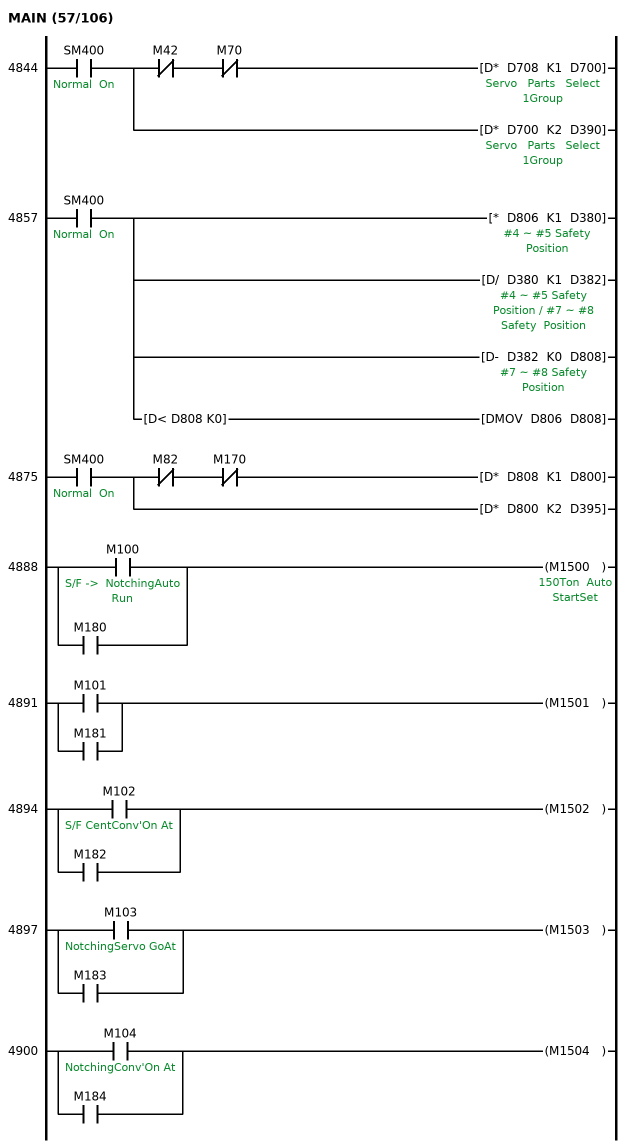
[picture p336: ladder of MAIN, rungs at steps 4844 to 4900]
4844  LD      SM400  ; Normal  On
      MPS
      ANI     M42
      ANI     M70
      D*      D708 K1 D700  ; Servo   Parts   Select  1Group
      MPP
      D*      D700 K2 D390
4857  LD      SM400  ; Normal  On
      *       D806 K1 D380  ; #4 ~ #5 Safety  Position
      D/      D380 K1 D382  ; #7 ~ #8 Safety  Position
      D-      D382 K0 D808
      ANDD<   D808 K0
      DMOV    D806 D808
4875  LD      SM400  ; Normal  On
      MPS
      ANI     M82
      ANI     M170
      D*      D808 K1 D800
      MPP
      D*      D800 K2 D395
4888  LD      M100  ; S/F ->  NotchingAuto Run
      OR      M180
      OUT     M1500  ; 150Ton  Auto    StartSet
4891  LD      M101
      OR      M181
      OUT     M1501
4894  LD      M102  ; S/F CentConv'On At
      OR      M182
      OUT     M1502
4897  LD      M103  ; NotchingServo GoAt
      OR      M183
      OUT     M1503
4900  LD      M104  ; NotchingConv'On At
      OR      M184
      OUT     M1504
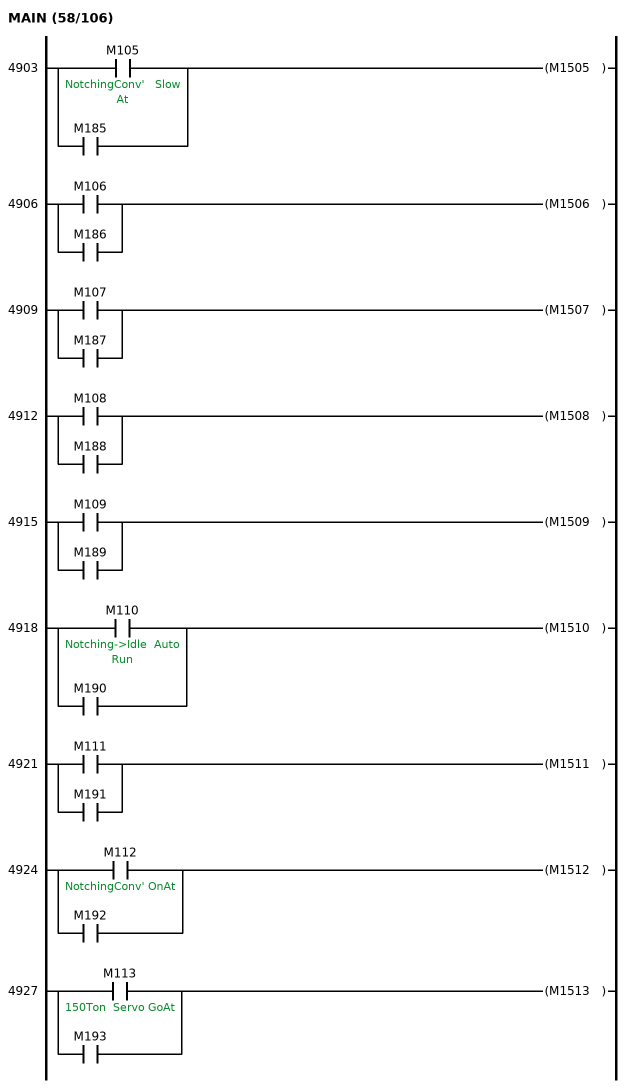
4903  LD      M105  ; NotchingConv'   Slow At
      OR      M185
      OUT     M1505
4906  LD      M106
      OR      M186
      OUT     M1506
4909  LD      M107
      OR      M187
      OUT     M1507
4912  LD      M108
      OR      M188
      OUT     M1508
4915  LD      M109
      OR      M189
      OUT     M1509
4918  LD      M110  ; Notching->Idle  Auto Run
      OR      M190
      OUT     M1510
4921  LD      M111
      OR      M191
      OUT     M1511
4924  LD      M112  ; NotchingConv' OnAt
      OR      M192
      OUT     M1512
4927  LD      M113  ; 150Ton  Servo GoAt
      OR      M193
      OUT     M1513
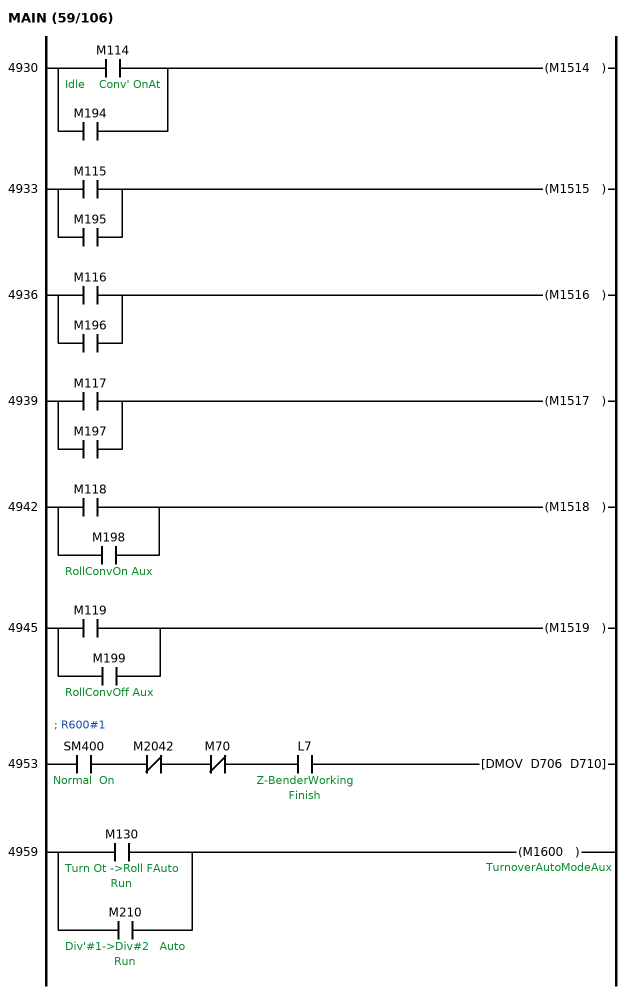
4930  LD      M114  ; Idle    Conv' OnAt
      OR      M194
      OUT     M1514
4933  LD      M115
      OR      M195
      OUT     M1515
4936  LD      M116
      OR      M196
      OUT     M1516
4939  LD      M117
      OR      M197
      OUT     M1517
4942  LD      M118
      OR      M198  ; RollConvOn Aux
      OUT     M1518
4945  LD      M119
      OR      M199  ; RollConvOff Aux
      OUT     M1519
; R600#1
4953  LD      SM400  ; Normal  On
      ANI     M2042
      ANI     M70
      AND     L7  ; Z-BenderWorking Finish
      DMOV    D706 D710
4959  LD      M130  ; Turn Ot ->Roll FAuto Run
      OR      M210  ; Div'#1->Div#2   Auto Run
      OUT     M1600  ; TurnoverAutoModeAux
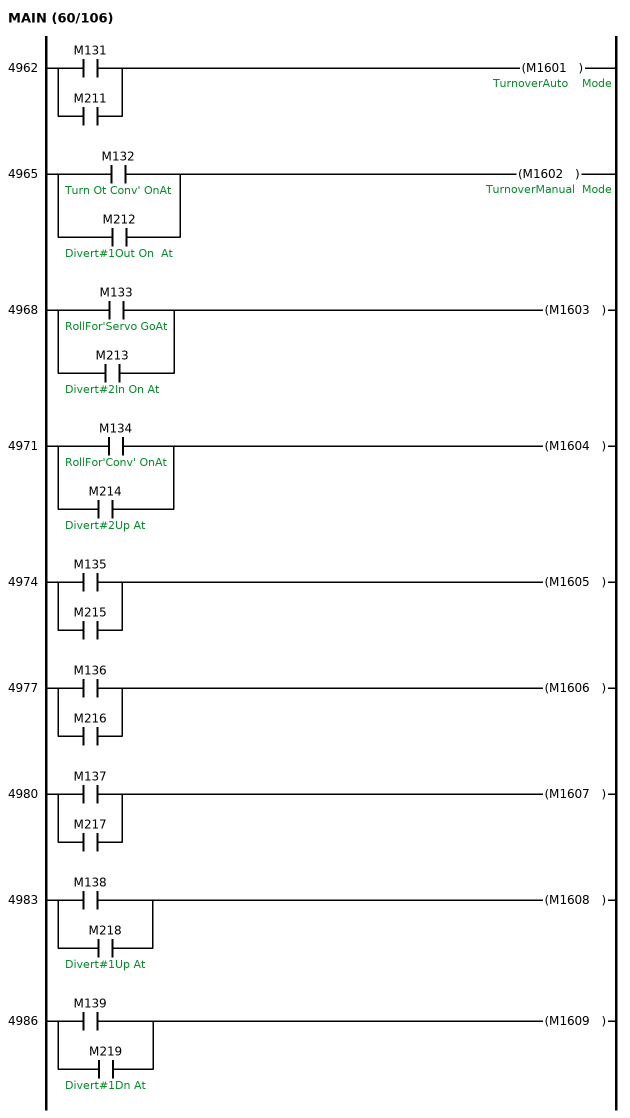
4962  LD      M131
      OR      M211
      OUT     M1601  ; TurnoverAuto    Mode
4965  LD      M132  ; Turn Ot Conv' OnAt
      OR      M212  ; Divert#1Out On  At
      OUT     M1602  ; TurnoverManual  Mode
4968  LD      M133  ; RollFor'Servo GoAt
      OR      M213  ; Divert#2In On At
      OUT     M1603
4971  LD      M134  ; RollFor'Conv' OnAt
      OR      M214  ; Divert#2Up At
      OUT     M1604
4974  LD      M135
      OR      M215
      OUT     M1605
4977  LD      M136
      OR      M216
      OUT     M1606
4980  LD      M137
      OR      M217
      OUT     M1607
4983  LD      M138
      OR      M218  ; Divert#1Up At
      OUT     M1608
4986  LD      M139
      OR      M219  ; Divert#1Dn At
      OUT     M1609
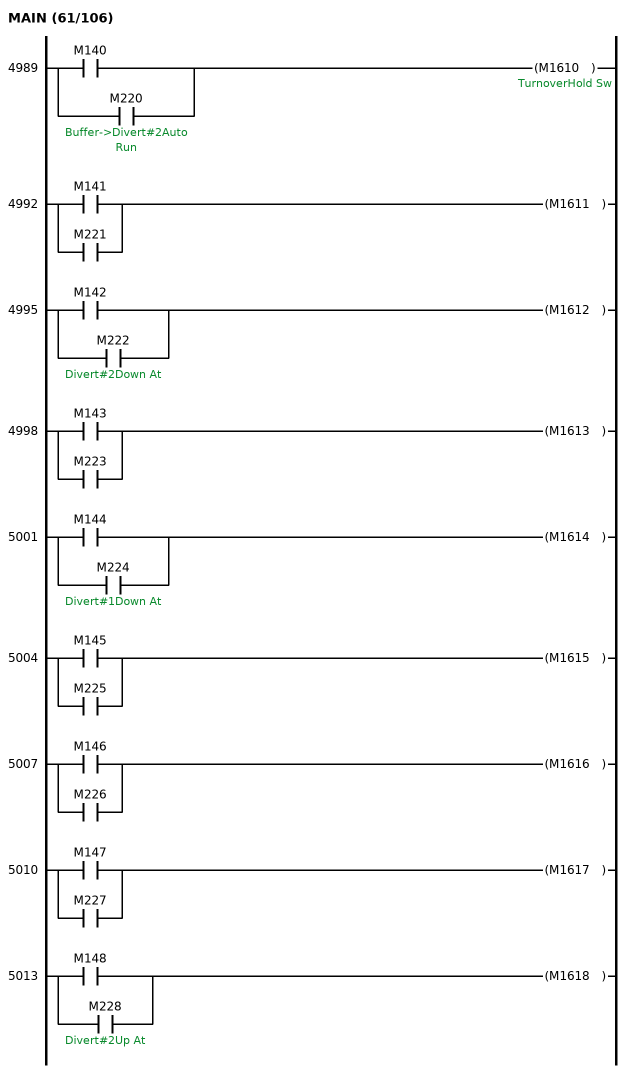
4989  LD      M140
      OR      M220  ; Buffer->Divert#2Auto Run
      OUT     M1610  ; TurnoverHold Sw
4992  LD      M141
      OR      M221
      OUT     M1611
4995  LD      M142
      OR      M222  ; Divert#2Down At
      OUT     M1612
4998  LD      M143
      OR      M223
      OUT     M1613
5001  LD      M144
      OR      M224  ; Divert#1Down At
      OUT     M1614
5004  LD      M145
      OR      M225
      OUT     M1615
5007  LD      M146
      OR      M226
      OUT     M1616
5010  LD      M147
      OR      M227
      OUT     M1617
5013  LD      M148
      OR      M228  ; Divert#2Up At
      OUT     M1618
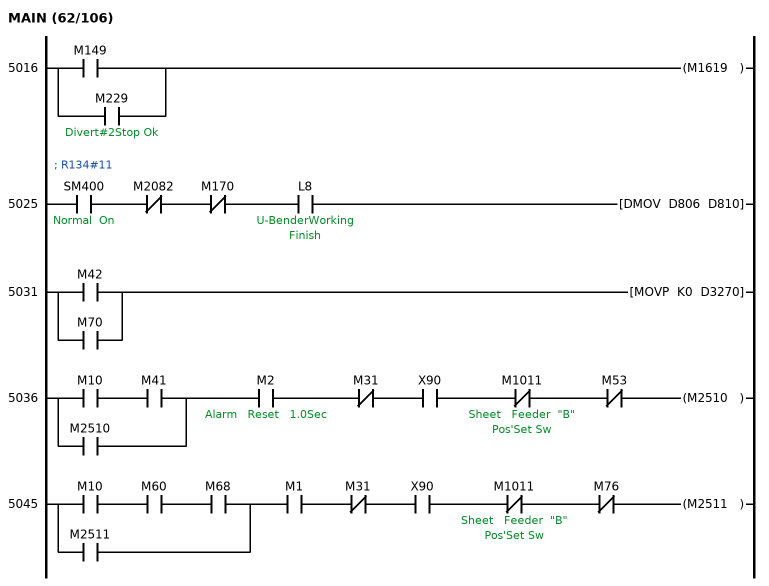
5016  LD      M149
      OR      M229  ; Divert#2Stop Ok
      OUT     M1619
; R134#11
5025  LD      SM400  ; Normal  On
      ANI     M2082
      ANI     M170
      AND     L8  ; U-BenderWorking Finish
      DMOV    D806 D810
5031  LD      M42
      OR      M70
      MOVP    K0 D3270
5036  LD      M10
      AND     M41
      OR      M2510
      AND     M2  ; Alarm   Reset   1.0Sec
      ANI     M31
      AND     X90
      ANI     M1011  ; Sheet   Feeder  "B" Pos'Set Sw
      ANI     M53
      OUT     M2510
5045  LD      M10
      AND     M60
      AND     M68
      OR      M2511
      AND     M1
      ANI     M31
      AND     X90
      ANI     M1011  ; Sheet   Feeder  "B" Pos'Set Sw
      ANI     M76
      OUT     M2511
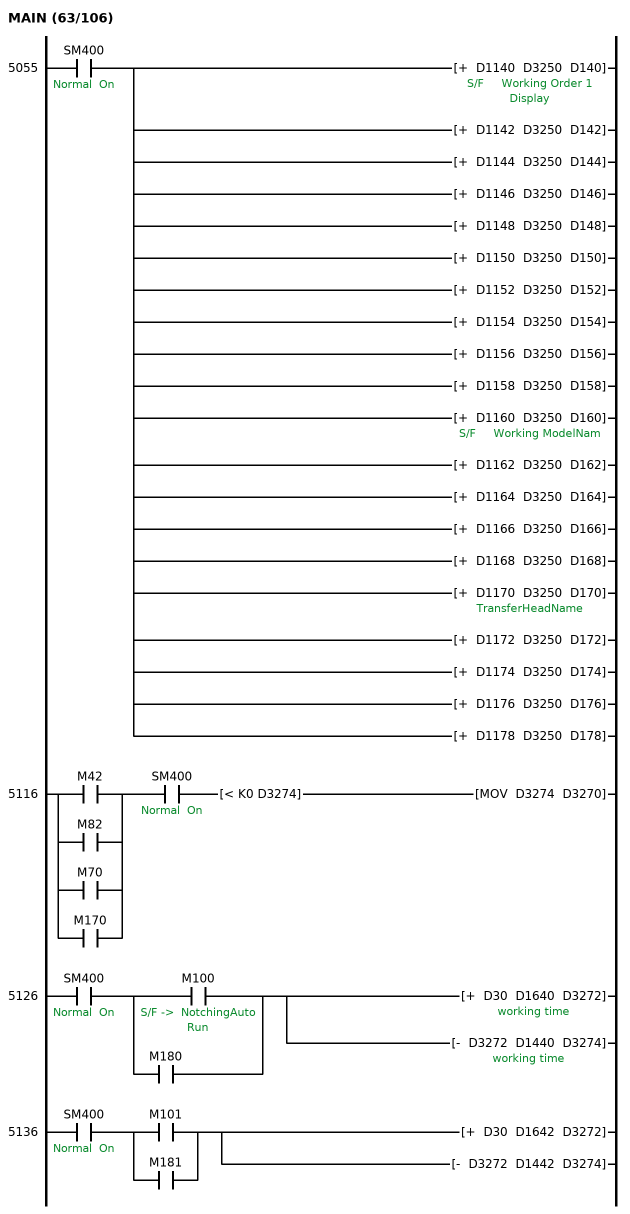
5055  LD      SM400  ; Normal  On
      +       D1140 D3250 D140
      +       D1142 D3250 D142
      +       D1144 D3250 D144
      +       D1146 D3250 D146
      +       D1148 D3250 D148
      +       D1150 D3250 D150
      +       D1152 D3250 D152
      +       D1154 D3250 D154
      +       D1156 D3250 D156
      +       D1158 D3250 D158
      +       D1160 D3250 D160
      +       D1162 D3250 D162
      +       D1164 D3250 D164
      +       D1166 D3250 D166
      +       D1168 D3250 D168
      +       D1170 D3250 D170
      +       D1172 D3250 D172
      +       D1174 D3250 D174
      +       D1176 D3250 D176
      +       D1178 D3250 D178
5116  LD      M42
      OR      M82
      OR      M70
      OR      M170
      AND     SM400  ; Normal  On
      AND<    K0 D3274
      MOV     D3274 D3270
5126  LD      SM400  ; Normal  On
      LD      M100  ; S/F ->  NotchingAuto Run
      OR      M180
      ANB
      +       D30 D1640 D3272  ; working time
      -       D3272 D1440 D3274
5136  LD      SM400  ; Normal  On
      LD      M101
      OR      M181
      ANB
      +       D30 D1642 D3272
      -       D3272 D1442 D3274
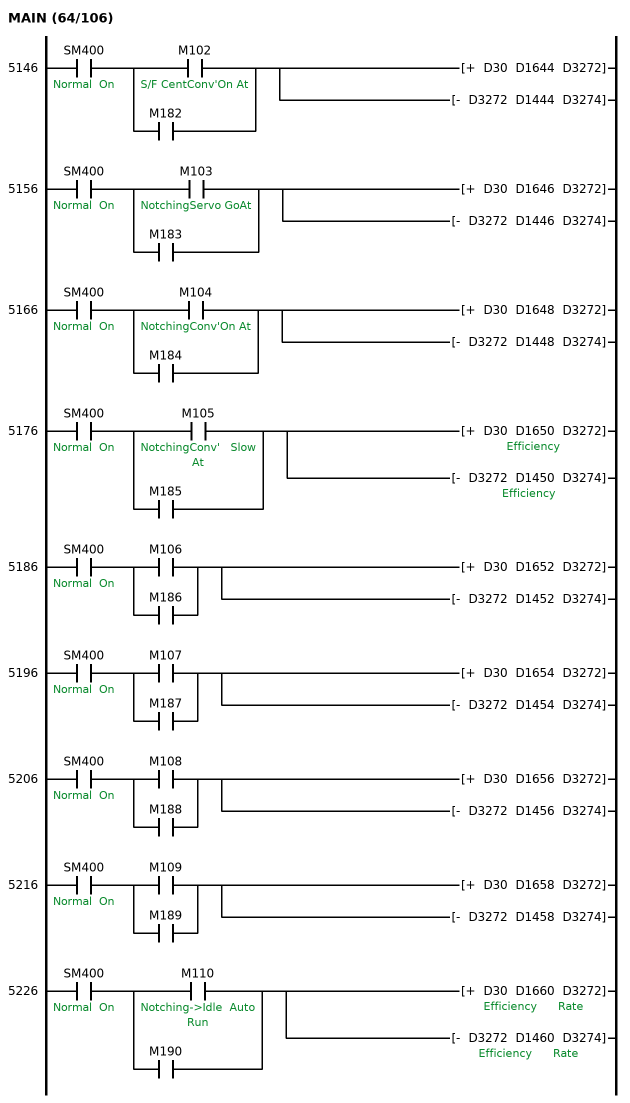
5146  LD      SM400  ; Normal  On
      LD      M102  ; S/F CentConv'On At
      OR      M182
      ANB
      +       D30 D1644 D3272
      -       D3272 D1444 D3274
5156  LD      SM400  ; Normal  On
      LD      M103  ; NotchingServo GoAt
      OR      M183
      ANB
      +       D30 D1646 D3272
      -       D3272 D1446 D3274
5166  LD      SM400  ; Normal  On
      LD      M104  ; NotchingConv'On At
      OR      M184
      ANB
      +       D30 D1648 D3272
      -       D3272 D1448 D3274
5176  LD      SM400  ; Normal  On
      LD      M105  ; NotchingConv'   Slow At
      OR      M185
      ANB
      +       D30 D1650 D3272  ; Efficiency
      -       D3272 D1450 D3274
5186  LD      SM400  ; Normal  On
      LD      M106
      OR      M186
      ANB
      +       D30 D1652 D3272
      -       D3272 D1452 D3274
5196  LD      SM400  ; Normal  On
      LD      M107
      OR      M187
      ANB
      +       D30 D1654 D3272
      -       D3272 D1454 D3274
5206  LD      SM400  ; Normal  On
      LD      M108
      OR      M188
      ANB
      +       D30 D1656 D3272
      -       D3272 D1456 D3274
5216  LD      SM400  ; Normal  On
      LD      M109
      OR      M189
      ANB
      +       D30 D1658 D3272
      -       D3272 D1458 D3274
5226  LD      SM400  ; Normal  On
      LD      M110  ; Notching->Idle  Auto Run
      OR      M190
      ANB
      +       D30 D1660 D3272  ; Efficiency      Rate
      -       D3272 D1460 D3274
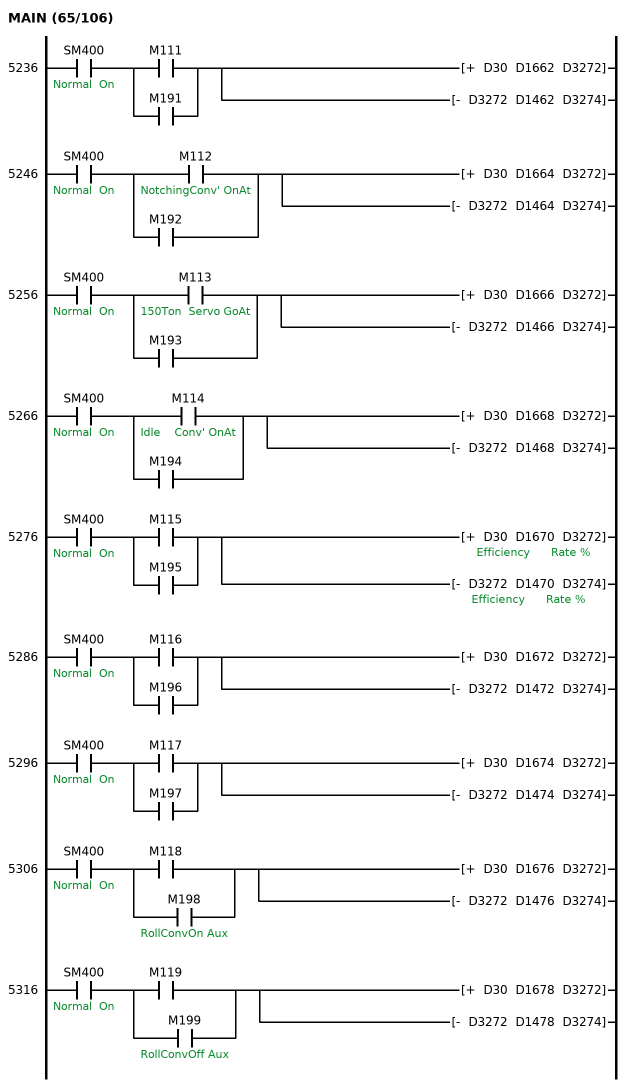
5236  LD      SM400  ; Normal  On
      LD      M111
      OR      M191
      ANB
      +       D30 D1662 D3272
      -       D3272 D1462 D3274
5246  LD      SM400  ; Normal  On
      LD      M112  ; NotchingConv' OnAt
      OR      M192
      ANB
      +       D30 D1664 D3272
      -       D3272 D1464 D3274
5256  LD      SM400  ; Normal  On
      LD      M113  ; 150Ton  Servo GoAt
      OR      M193
      ANB
      +       D30 D1666 D3272
      -       D3272 D1466 D3274
5266  LD      SM400  ; Normal  On
      LD      M114  ; Idle    Conv' OnAt
      OR      M194
      ANB
      +       D30 D1668 D3272
      -       D3272 D1468 D3274
5276  LD      SM400  ; Normal  On
      LD      M115
      OR      M195
      ANB
      +       D30 D1670 D3272  ; Efficiency      Rate %
      -       D3272 D1470 D3274
5286  LD      SM400  ; Normal  On
      LD      M116
      OR      M196
      ANB
      +       D30 D1672 D3272
      -       D3272 D1472 D3274
5296  LD      SM400  ; Normal  On
      LD      M117
      OR      M197
      ANB
      +       D30 D1674 D3272
      -       D3272 D1474 D3274
5306  LD      SM400  ; Normal  On
      LD      M118
      OR      M198  ; RollConvOn Aux
      ANB
      +       D30 D1676 D3272
      -       D3272 D1476 D3274
5316  LD      SM400  ; Normal  On
      LD      M119
      OR      M199  ; RollConvOff Aux
      ANB
      +       D30 D1678 D3272
      -       D3272 D1478 D3274
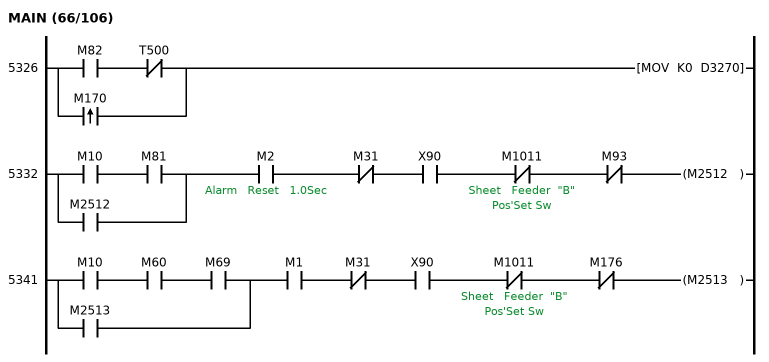
5326  LD      M82
      ANI     T500
      ORP     M170
      MOV     K0 D3270
5332  LD      M10
      AND     M81
      OR      M2512
      AND     M2  ; Alarm   Reset   1.0Sec
      ANI     M31
      AND     X90
      ANI     M1011  ; Sheet   Feeder  "B" Pos'Set Sw
      ANI     M93
      OUT     M2512
5341  LD      M10
      AND     M60
      AND     M69
      OR      M2513
      AND     M1
      ANI     M31
      AND     X90
      ANI     M1011  ; Sheet   Feeder  "B" Pos'Set Sw
      ANI     M176
      OUT     M2513
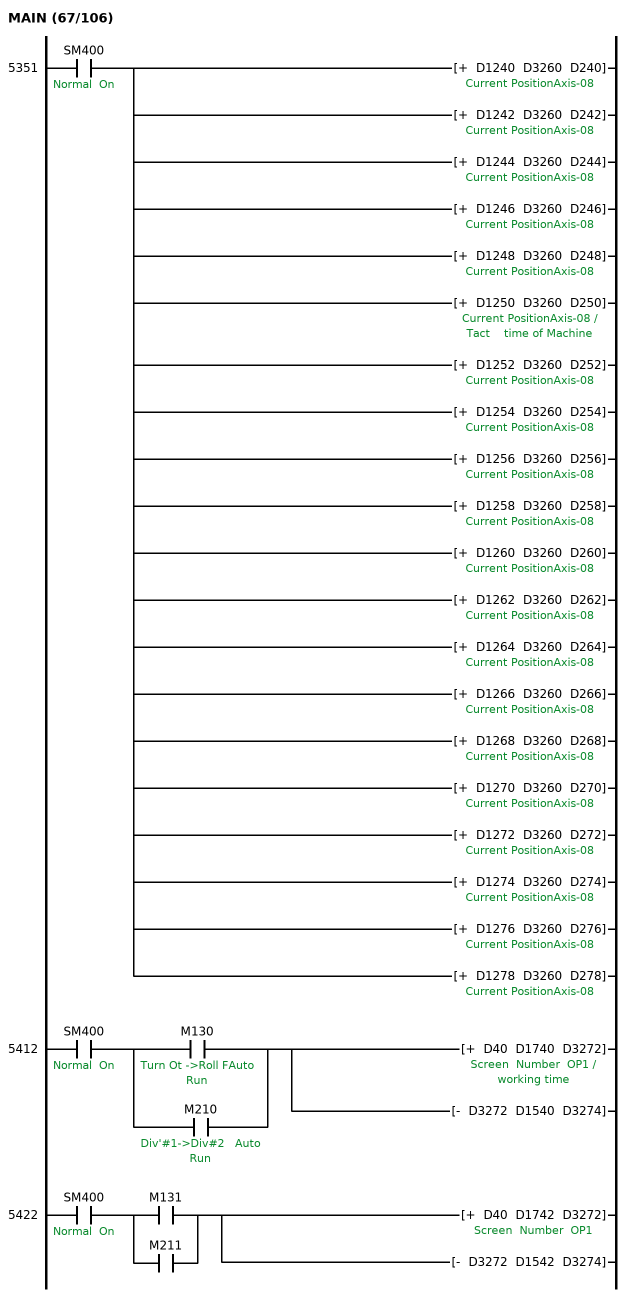
5351  LD      SM400  ; Normal  On
      +       D1240 D3260 D240  ; Current PositionAxis-08
      +       D1242 D3260 D242
      +       D1244 D3260 D244
      +       D1246 D3260 D246
      +       D1248 D3260 D248
      +       D1250 D3260 D250
      +       D1252 D3260 D252
      +       D1254 D3260 D254
      +       D1256 D3260 D256
      +       D1258 D3260 D258
      +       D1260 D3260 D260
      +       D1262 D3260 D262
      +       D1264 D3260 D264
      +       D1266 D3260 D266
      +       D1268 D3260 D268
      +       D1270 D3260 D270
      +       D1272 D3260 D272
      +       D1274 D3260 D274
      +       D1276 D3260 D276
      +       D1278 D3260 D278
5412  LD      SM400  ; Normal  On
      LD      M130  ; Turn Ot ->Roll FAuto Run
      OR      M210  ; Div'#1->Div#2   Auto Run
      ANB
      +       D40 D1740 D3272  ; working time
      -       D3272 D1540 D3274
5422  LD      SM400  ; Normal  On
      LD      M131
      OR      M211
      ANB
      +       D40 D1742 D3272
      -       D3272 D1542 D3274
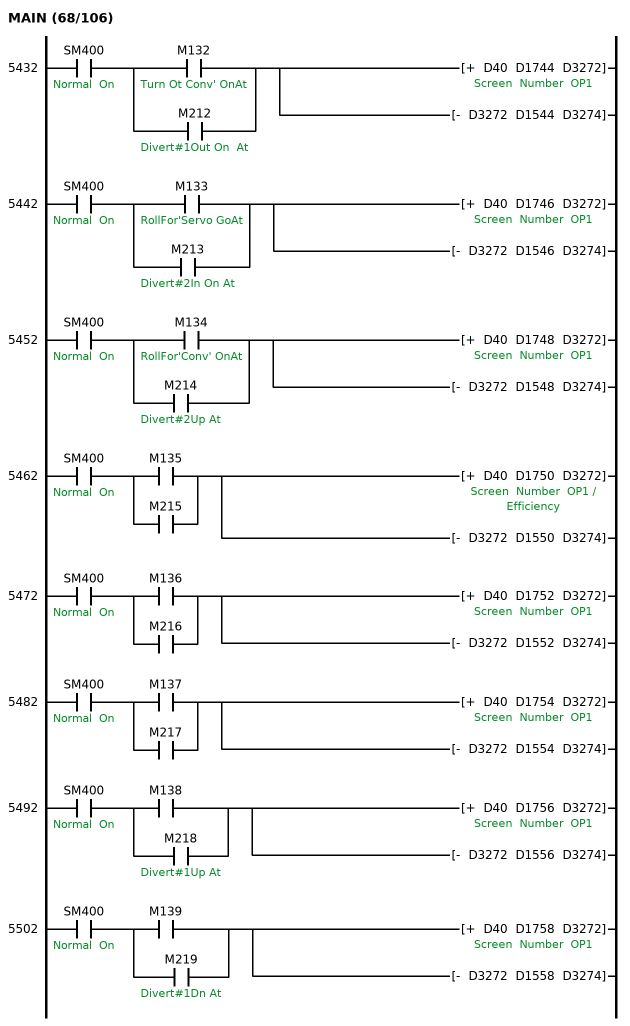
5432  LD      SM400  ; Normal  On
      LD      M132  ; Turn Ot Conv' OnAt
      OR      M212  ; Divert#1Out On  At
      ANB
      +       D40 D1744 D3272
      -       D3272 D1544 D3274
5442  LD      SM400  ; Normal  On
      LD      M133  ; RollFor'Servo GoAt
      OR      M213  ; Divert#2In On At
      ANB
      +       D40 D1746 D3272
      -       D3272 D1546 D3274
5452  LD      SM400  ; Normal  On
      LD      M134  ; RollFor'Conv' OnAt
      OR      M214  ; Divert#2Up At
      ANB
      +       D40 D1748 D3272
      -       D3272 D1548 D3274
5462  LD      SM400  ; Normal  On
      LD      M135
      OR      M215
      ANB
      +       D40 D1750 D3272  ; Efficiency
      -       D3272 D1550 D3274
5472  LD      SM400  ; Normal  On
      LD      M136
      OR      M216
      ANB
      +       D40 D1752 D3272
      -       D3272 D1552 D3274
5482  LD      SM400  ; Normal  On
      LD      M137
      OR      M217
      ANB
      +       D40 D1754 D3272
      -       D3272 D1554 D3274
5492  LD      SM400  ; Normal  On
      LD      M138
      OR      M218  ; Divert#1Up At
      ANB
      +       D40 D1756 D3272
      -       D3272 D1556 D3274
5502  LD      SM400  ; Normal  On
      LD      M139
      OR      M219  ; Divert#1Dn At
      ANB
      +       D40 D1758 D3272
      -       D3272 D1558 D3274
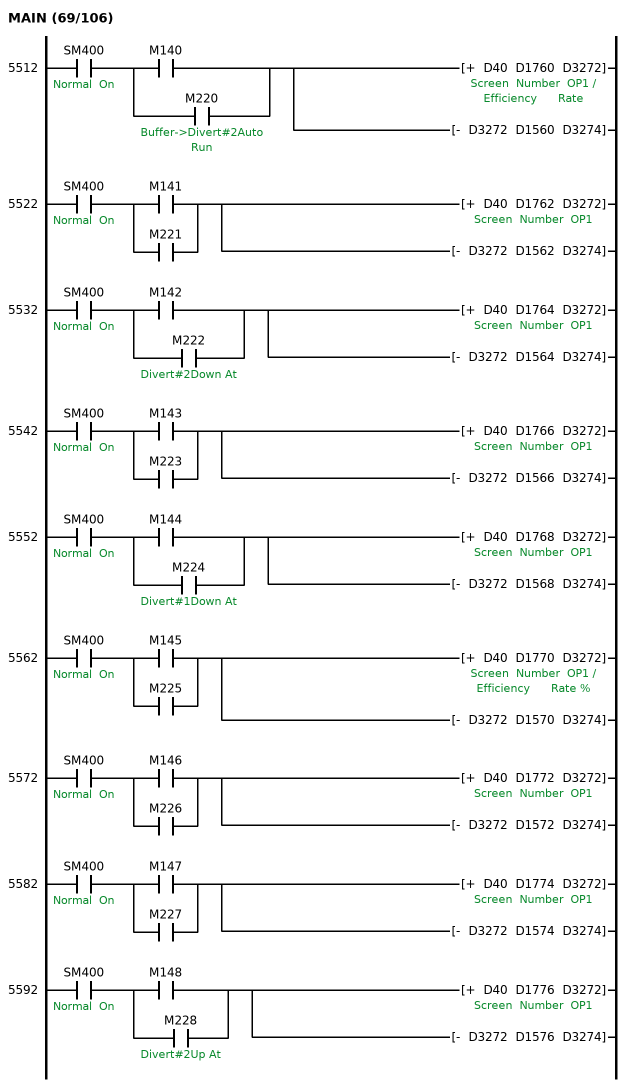
5512  LD      SM400  ; Normal  On
      LD      M140
      OR      M220  ; Buffer->Divert#2Auto Run
      ANB
      +       D40 D1760 D3272  ; Efficiency      Rate
      -       D3272 D1560 D3274
5522  LD      SM400  ; Normal  On
      LD      M141
      OR      M221
      ANB
      +       D40 D1762 D3272
      -       D3272 D1562 D3274
5532  LD      SM400  ; Normal  On
      LD      M142
      OR      M222  ; Divert#2Down At
      ANB
      +       D40 D1764 D3272
      -       D3272 D1564 D3274
5542  LD      SM400  ; Normal  On
      LD      M143
      OR      M223
      ANB
      +       D40 D1766 D3272
      -       D3272 D1566 D3274
5552  LD      SM400  ; Normal  On
      LD      M144
      OR      M224  ; Divert#1Down At
      ANB
      +       D40 D1768 D3272
      -       D3272 D1568 D3274
5562  LD      SM400  ; Normal  On
      LD      M145
      OR      M225
      ANB
      +       D40 D1770 D3272  ; Efficiency      Rate %
      -       D3272 D1570 D3274
5572  LD      SM400  ; Normal  On
      LD      M146
      OR      M226
      ANB
      +       D40 D1772 D3272
      -       D3272 D1572 D3274
5582  LD      SM400  ; Normal  On
      LD      M147
      OR      M227
      ANB
      +       D40 D1774 D3272
      -       D3272 D1574 D3274
5592  LD      SM400  ; Normal  On
      LD      M148
      OR      M228  ; Divert#2Up At
      ANB
      +       D40 D1776 D3272
      -       D3272 D1576 D3274
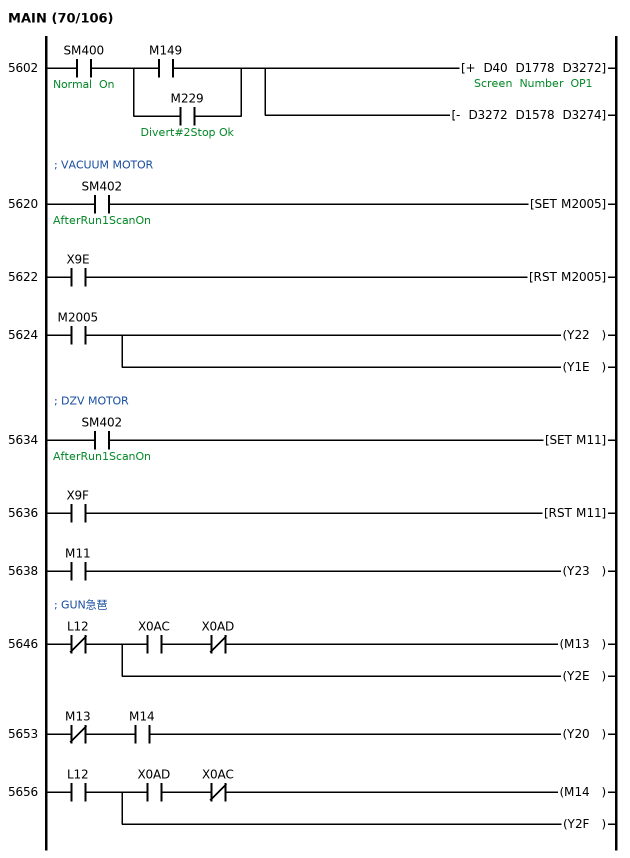
5602  LD      SM400  ; Normal  On
      LD      M149
      OR      M229  ; Divert#2Stop Ok
      ANB
      +       D40 D1778 D3272
      -       D3272 D1578 D3274
; VACUUM MOTOR
5620  LD      SM402  ; AfterRun1ScanOn
      SET     M2005
5622  LD      X9E
      RST     M2005
5624  LD      M2005
      OUT     Y22
      OUT     Y1E
; DZV MOTOR
5634  LD      SM402  ; AfterRun1ScanOn
      SET     M11
5636  LD      X9F
      RST     M11
5638  LD      M11
      OUT     Y23
; GUN선택
5646  LDI     L12
      MPS
      AND     X0AC
      ANI     X0AD
      OUT     M13
      MPP
      OUT     Y2E
5653  LDI     M13
      AND     M14
      OUT     Y20
5656  LD      L12
      MPS
      AND     X0AD
      ANI     X0AC
      OUT     M14
      MPP
      OUT     Y2F
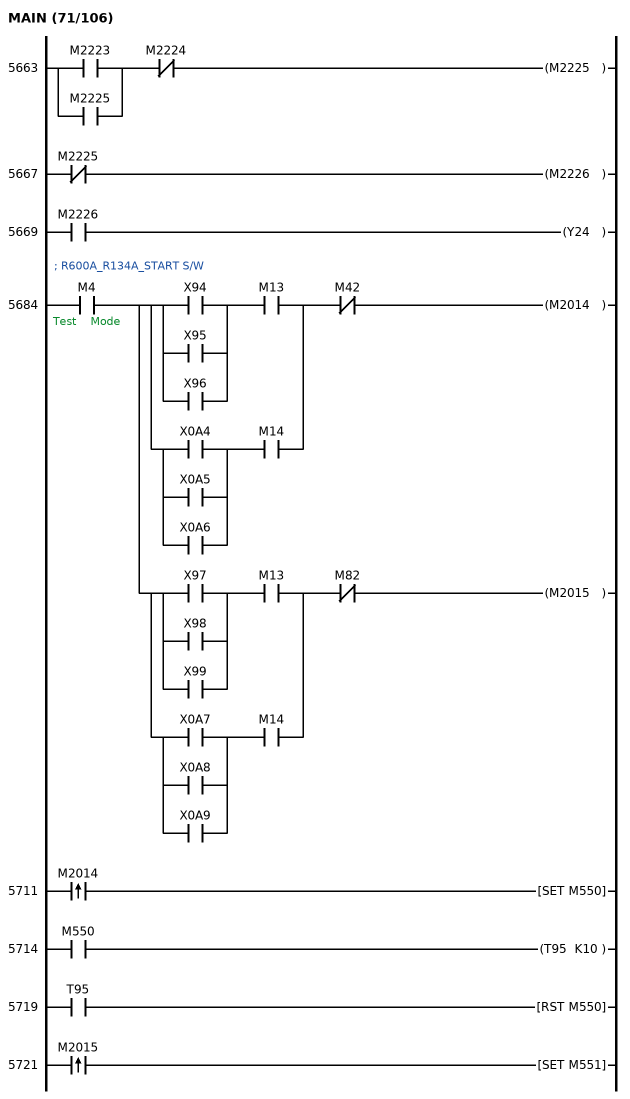
5663  LD      M2223
      OR      M2225
      ANI     M2224
      OUT     M2225
5667  LDI     M2225
      OUT     M2226
5669  LD      M2226
      OUT     Y24
; R600A_R134A_START S/W
5684  LD      M4  ; Test    Mode
      MPS
      LD      X94
      OR      X95
      OR      X96
      AND     M13
      LD      X0A4
      OR      X0A5
      OR      X0A6
      AND     M14
      ORB
      ANB
      ANI     M42
      OUT     M2014
      MPP
      LD      X97
      OR      X98
      OR      X99
      AND     M13
      LD      X0A7
      OR      X0A8
      OR      X0A9
      AND     M14
      ORB
      ANB
      ANI     M82
      OUT     M2015
5711  LDP     M2014
      SET     M550
5714  LD      M550
      OUT     T95 K10
5719  LD      T95
      RST     M550
5721  LDP     M2015
      SET     M551
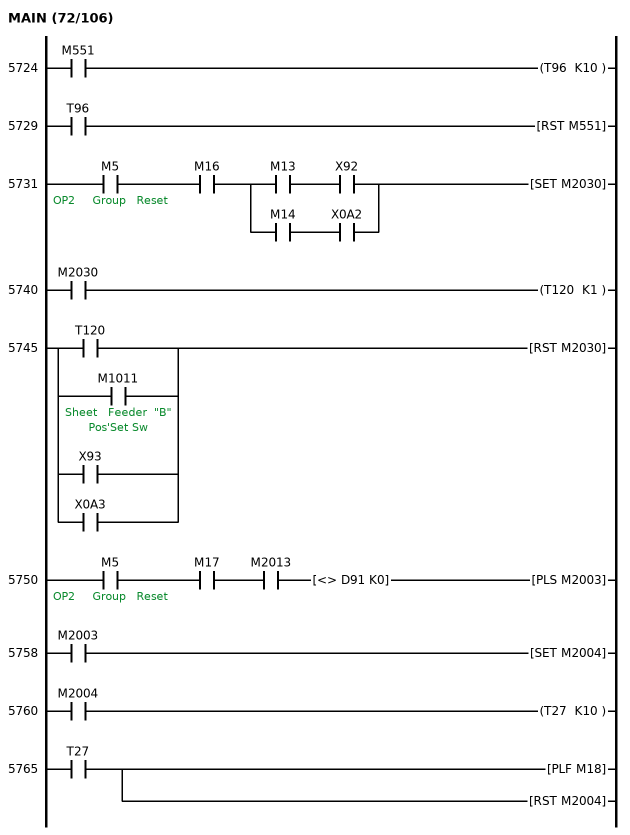
5724  LD      M551
      OUT     T96 K10
5729  LD      T96
      RST     M551
5731  LD      M5  ; OP2     Group   Reset
      AND     M16
      LD      M13
      AND     X92
      LD      M14
      AND     X0A2
      ORB
      ANB
      SET     M2030
5740  LD      M2030
      OUT     T120 K1
5745  LD      T120
      OR      M1011  ; Sheet   Feeder  "B" Pos'Set Sw
      OR      X93
      OR      X0A3
      RST     M2030
5750  LD      M5  ; OP2     Group   Reset
      AND     M17
      AND     M2013
      AND<>   D91 K0
      PLS     M2003
5758  LD      M2003
      SET     M2004
5760  LD      M2004
      OUT     T27 K10
5765  LD      T27
      PLF     M18
      RST     M2004
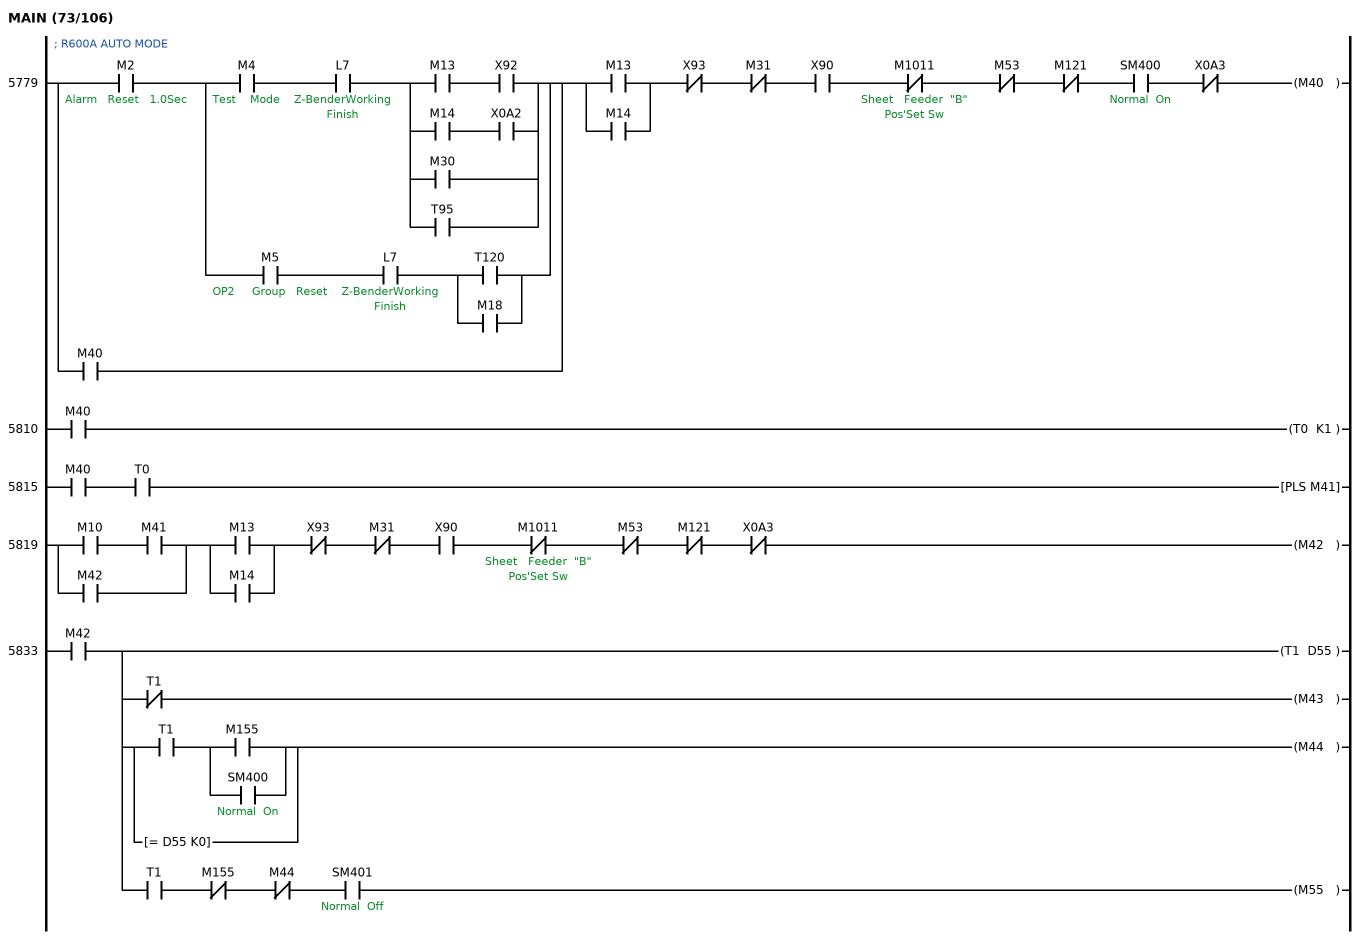
; R600A AUTO MODE
5779  LD      M2  ; Alarm   Reset   1.0Sec
      LD      M4  ; Test    Mode
      AND     L7  ; Z-BenderWorking Finish
      LD      M13
      AND     X92
      LD      M14
      AND     X0A2
      ORB
      OR      M30
      OR      T95
      ANB
      LD      M5  ; OP2     Group   Reset
      AND     L7  ; Z-BenderWorking Finish
      LD      T120
      OR      M18
      ANB
      ORB
      ANB
      OR      M40
      LD      M13
      OR      M14
      ANB
      ANI     X93
      ANI     M31
      AND     X90
      ANI     M1011  ; Sheet   Feeder  "B" Pos'Set Sw
      ANI     M53
      ANI     M121
      AND     SM400  ; Normal  On
      ANI     X0A3
      OUT     M40
5810  LD      M40
      OUT     T0 K1
5815  LD      M40
      AND     T0
      PLS     M41
5819  LD      M10
      AND     M41
      OR      M42
      LD      M13
      OR      M14
      ANB
      ANI     X93
      ANI     M31
      AND     X90
      ANI     M1011  ; Sheet   Feeder  "B" Pos'Set Sw
      ANI     M53
      ANI     M121
      ANI     X0A3
      OUT     M42
5833  LD      M42
      OUT     T1 D55
      MPS
      ANI     T1
      OUT     M43
      MRD
      LD      T1
      LD      M155
      OR      SM400  ; Normal  On
      ANB
      OR=     D55 K0
      ANB
      OUT     M44
      MPP
      AND     T1
      ANI     M155
      ANI     M44
      AND     SM401  ; Normal  Off
      OUT     M55
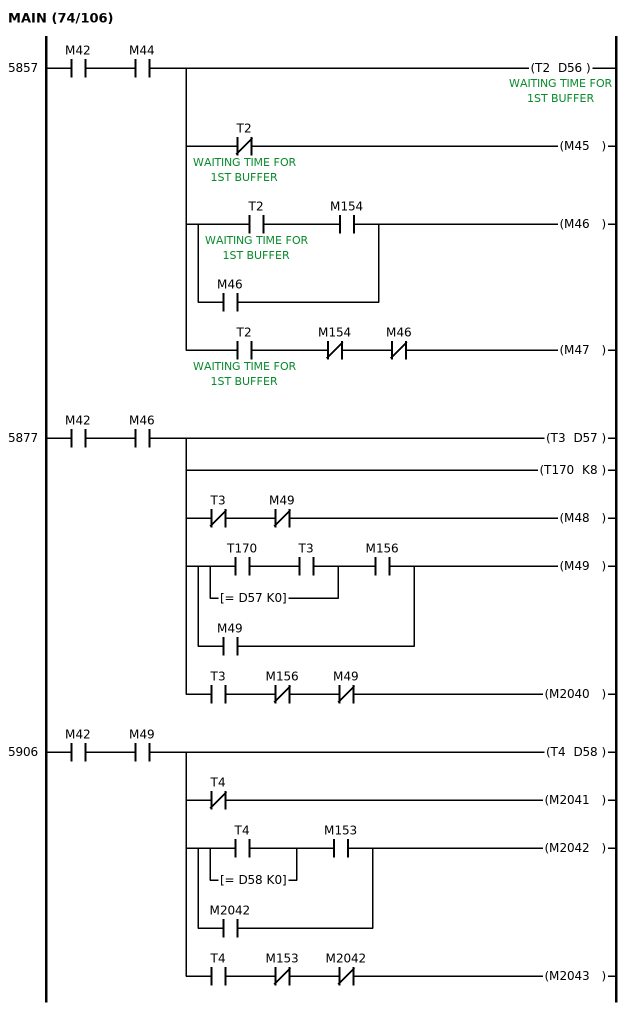
5857  LD      M42
      AND     M44
      OUT     T2 D56  ; WAITING TIME FOR 1ST BUFFER
      MPS
      ANI     T2  ; WAITING TIME FOR 1ST BUFFER
      OUT     M45
      MRD
      LD      T2  ; WAITING TIME FOR 1ST BUFFER
      AND     M154
      OR      M46
      ANB
      OUT     M46
      MPP
      AND     T2  ; WAITING TIME FOR 1ST BUFFER
      ANI     M154
      ANI     M46
      OUT     M47
5877  LD      M42
      AND     M46
      OUT     T3 D57
      OUT     T170 K8
      MPS
      ANI     T3
      ANI     M49
      OUT     M48
      MRD
      LD      T170
      AND     T3
      OR=     D57 K0
      AND     M156
      OR      M49
      ANB
      OUT     M49
      MPP
      AND     T3
      ANI     M156
      ANI     M49
      OUT     M2040
5906  LD      M42
      AND     M49
      OUT     T4 D58
      MPS
      ANI     T4
      OUT     M2041
      MRD
      LD      T4
      OR=     D58 K0
      AND     M153
      OR      M2042
      ANB
      OUT     M2042
      MPP
      AND     T4
      ANI     M153
      ANI     M2042
      OUT     M2043
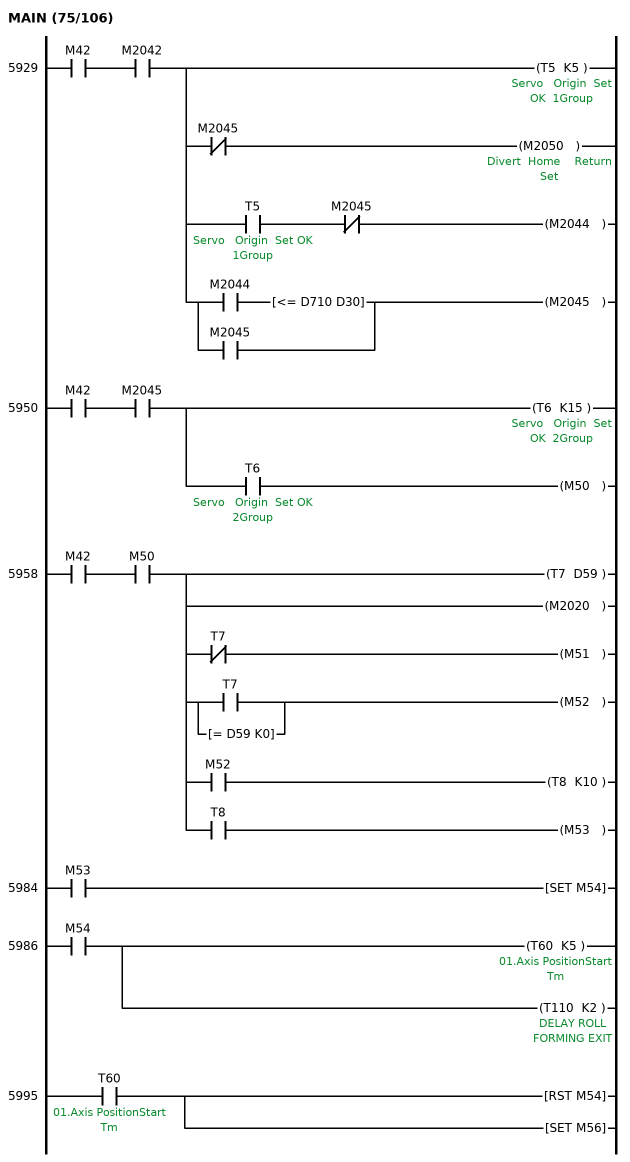
5929  LD      M42
      AND     M2042
      OUT     T5 K5  ; Servo   Origin  Set OK  1Group
      MPS
      ANI     M2045
      OUT     M2050  ; Divert  Home    Return  Set
      MRD
      AND     T5  ; Servo   Origin  Set OK  1Group
      ANI     M2045
      OUT     M2044
      MPP
      LD      M2044
      AND<=   D710 D30
      OR      M2045
      ANB
      OUT     M2045
5950  LD      M42
      AND     M2045
      OUT     T6 K15  ; Servo   Origin  Set OK  2Group
      AND     T6  ; Servo   Origin  Set OK  2Group
      OUT     M50
5958  LD      M42
      AND     M50
      OUT     T7 D59
      OUT     M2020
      MPS
      ANI     T7
      OUT     M51
      MRD
      LD      T7
      OR=     D59 K0
      ANB
      OUT     M52
      MRD
      AND     M52
      OUT     T8 K10
      MPP
      AND     T8
      OUT     M53
5984  LD      M53
      SET     M54
5986  LD      M54
      OUT     T60 K5  ; 01.Axis PositionStart Tm
      OUT     T110 K2  ; DELAY ROLL FORMING EXIT
5995  LD      T60  ; 01.Axis PositionStart Tm
      RST     M54
      SET     M56
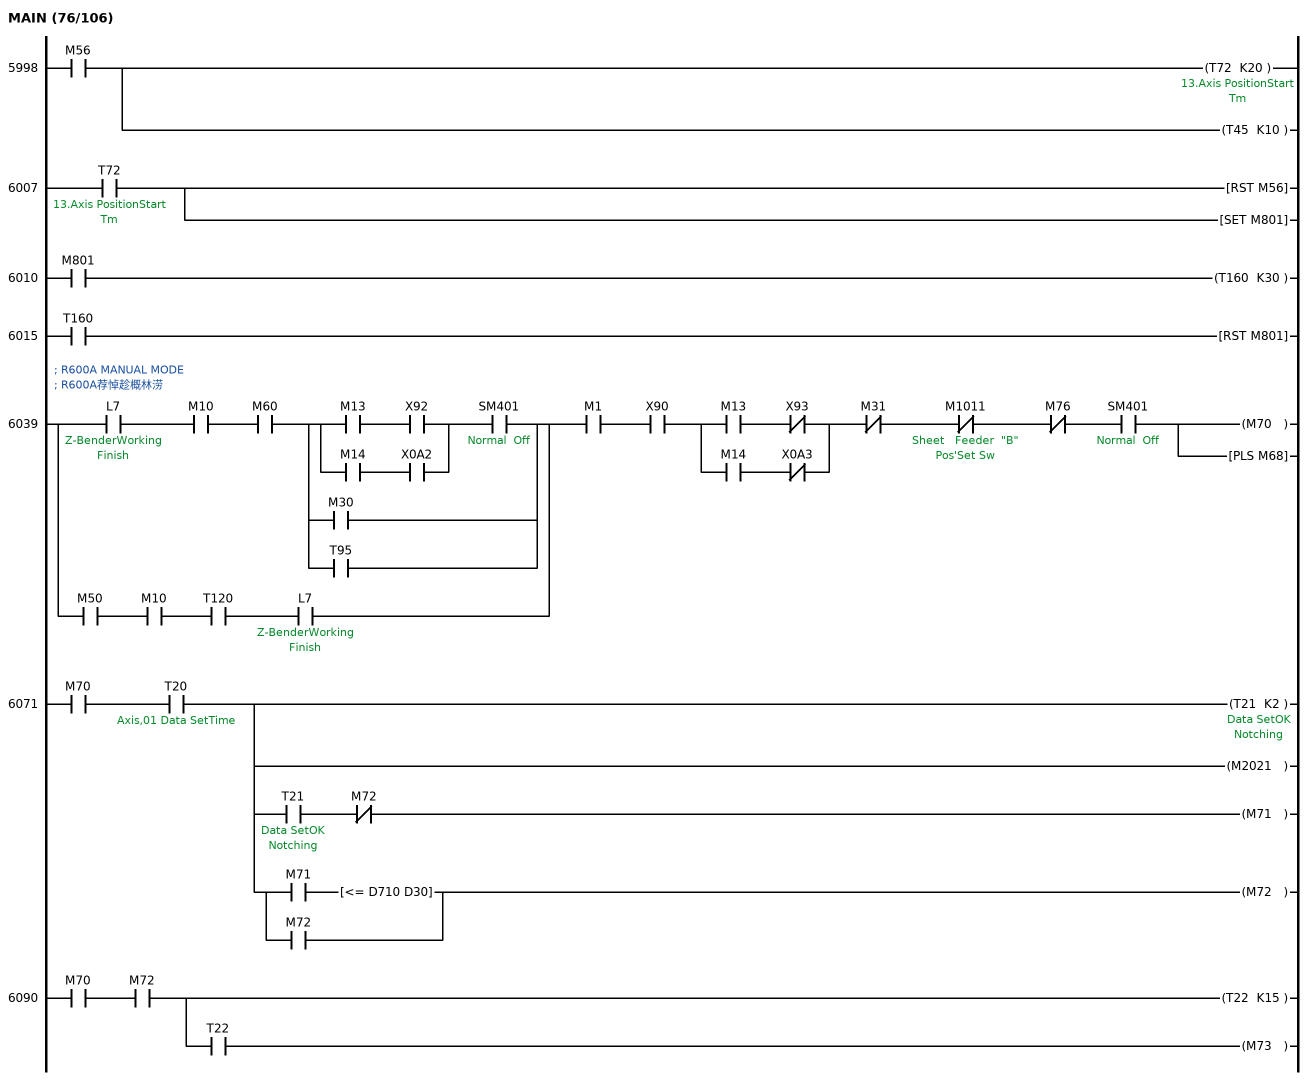
5998  LD      M56
      OUT     T72 K20  ; 13.Axis PositionStart Tm
      OUT     T45 K10
6007  LD      T72  ; 13.Axis PositionStart Tm
      RST     M56
      SET     M801
6010  LD      M801
      OUT     T160 K30
6015  LD      T160
      RST     M801
; R600A MANUAL MODE
; R600A수동냉매주입
6039  LD      L7  ; Z-BenderWorking Finish
      AND     M10
      AND     M60
      LD      M13
      AND     X92
      LD      M14
      AND     X0A2
      ORB
      AND     SM401  ; Normal  Off
      OR      M30
      OR      T95
      ANB
      LD      M50
      AND     M10
      AND     T120
      AND     L7  ; Z-BenderWorking Finish
      ORB
      AND     M1
      AND     X90
      LD      M13
      ANI     X93
      LD      M14
      ANI     X0A3
      ORB
      ANB
      ANI     M31
      ANI     M1011  ; Sheet   Feeder  "B" Pos'Set Sw
      ANI     M76
      AND     SM401  ; Normal  Off
      OUT     M70
      PLS     M68
6071  LD      M70
      AND     T20  ; Axis,01 Data SetTime
      OUT     T21 K2  ; Data SetOK      Notching
      OUT     M2021
      MPS
      AND     T21  ; Data SetOK      Notching
      ANI     M72
      OUT     M71
      MPP
      LD      M71
      AND<=   D710 D30
      OR      M72
      ANB
      OUT     M72
6090  LD      M70
      AND     M72
      OUT     T22 K15
      AND     T22
      OUT     M73
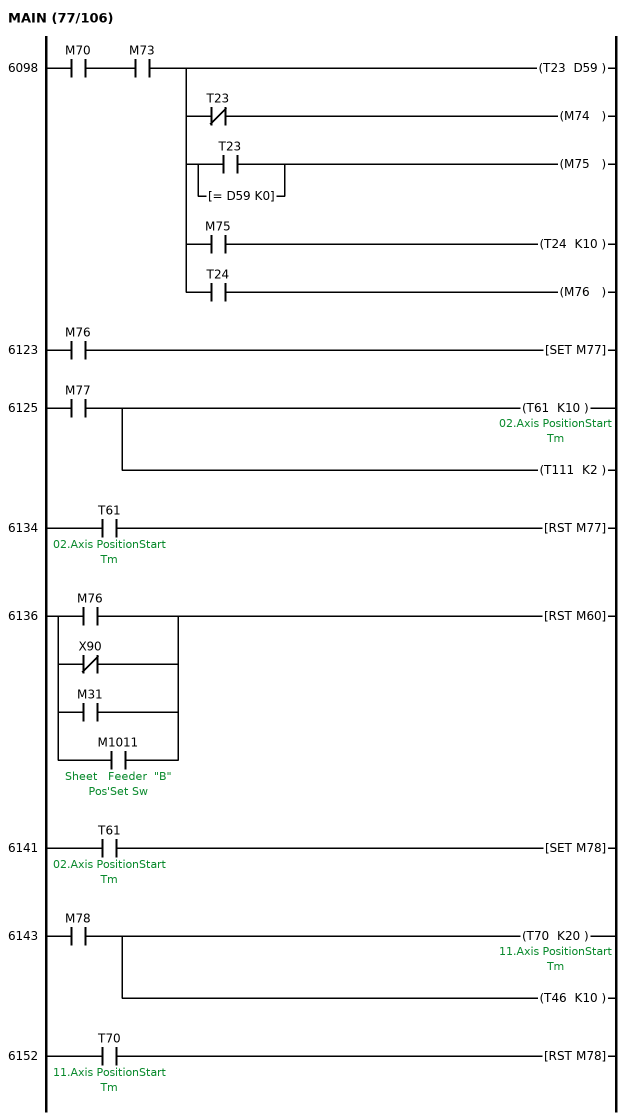
6098  LD      M70
      AND     M73
      OUT     T23 D59
      MPS
      ANI     T23
      OUT     M74
      MRD
      LD      T23
      OR=     D59 K0
      ANB
      OUT     M75
      MRD
      AND     M75
      OUT     T24 K10
      MPP
      AND     T24
      OUT     M76
6123  LD      M76
      SET     M77
6125  LD      M77
      OUT     T61 K10  ; 02.Axis PositionStart Tm
      OUT     T111 K2
6134  LD      T61  ; 02.Axis PositionStart Tm
      RST     M77
6136  LD      M76
      ORI     X90
      OR      M31
      OR      M1011  ; Sheet   Feeder  "B" Pos'Set Sw
      RST     M60
6141  LD      T61  ; 02.Axis PositionStart Tm
      SET     M78
6143  LD      M78
      OUT     T70 K20  ; 11.Axis PositionStart Tm
      OUT     T46 K10
6152  LD      T70  ; 11.Axis PositionStart Tm
      RST     M78
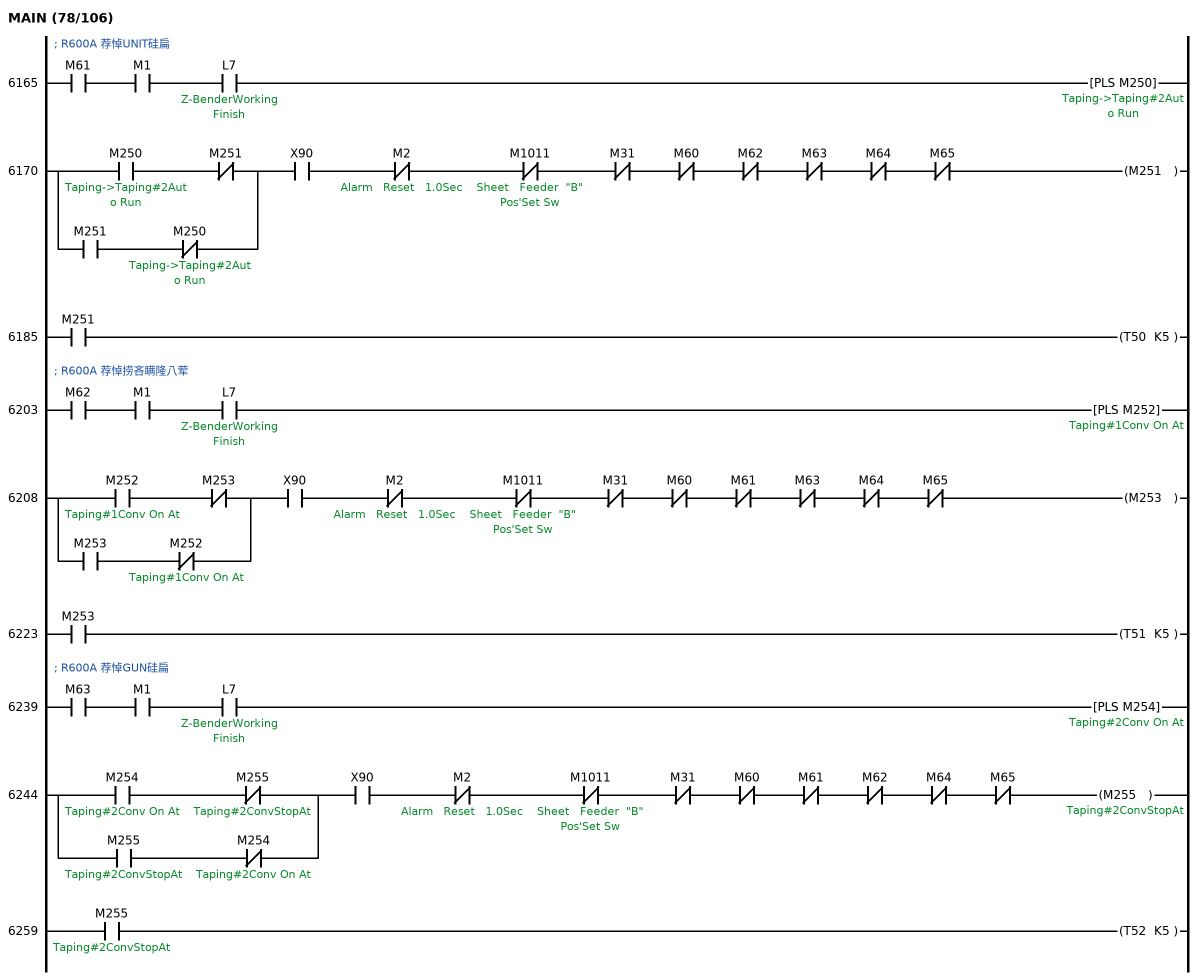
; R600A 수동UNIT배기
6165  LD      M61
      AND     M1
      AND     L7  ; Z-BenderWorking Finish
      PLS     M250  ; Taping->Taping#2Auto Run
6170  LD      M250  ; Taping->Taping#2Auto Run
      ANI     M251
      LD      M251
      ANI     M250  ; Taping->Taping#2Auto Run
      ORB
      AND     X90
      ANI     M2  ; Alarm   Reset   1.0Sec
      ANI     M1011  ; Sheet   Feeder  "B" Pos'Set Sw
      ANI     M31
      ANI     M60
      ANI     M62
      ANI     M63
      ANI     M64
      ANI     M65
      OUT     M251
6185  LD      M251
      OUT     T50 K5
; R600A 수동이중차징검사
6203  LD      M62
      AND     M1
      AND     L7  ; Z-BenderWorking Finish
      PLS     M252  ; Taping#1Conv On At
6208  LD      M252  ; Taping#1Conv On At
      ANI     M253
      LD      M253
      ANI     M252  ; Taping#1Conv On At
      ORB
      AND     X90
      ANI     M2  ; Alarm   Reset   1.0Sec
      ANI     M1011  ; Sheet   Feeder  "B" Pos'Set Sw
      ANI     M31
      ANI     M60
      ANI     M61
      ANI     M63
      ANI     M64
      ANI     M65
      OUT     M253
6223  LD      M253
      OUT     T51 K5
; R600A 수동GUN배기
6239  LD      M63
      AND     M1
      AND     L7  ; Z-BenderWorking Finish
      PLS     M254  ; Taping#2Conv On At
6244  LD      M254  ; Taping#2Conv On At
      ANI     M255  ; Taping#2ConvStopAt
      LD      M255  ; Taping#2ConvStopAt
      ANI     M254  ; Taping#2Conv On At
      ORB
      AND     X90
      ANI     M2  ; Alarm   Reset   1.0Sec
      ANI     M1011  ; Sheet   Feeder  "B" Pos'Set Sw
      ANI     M31
      ANI     M60
      ANI     M61
      ANI     M62
      ANI     M64
      ANI     M65
      OUT     M255  ; Taping#2ConvStopAt
6259  LD      M255  ; Taping#2ConvStopAt
      OUT     T52 K5
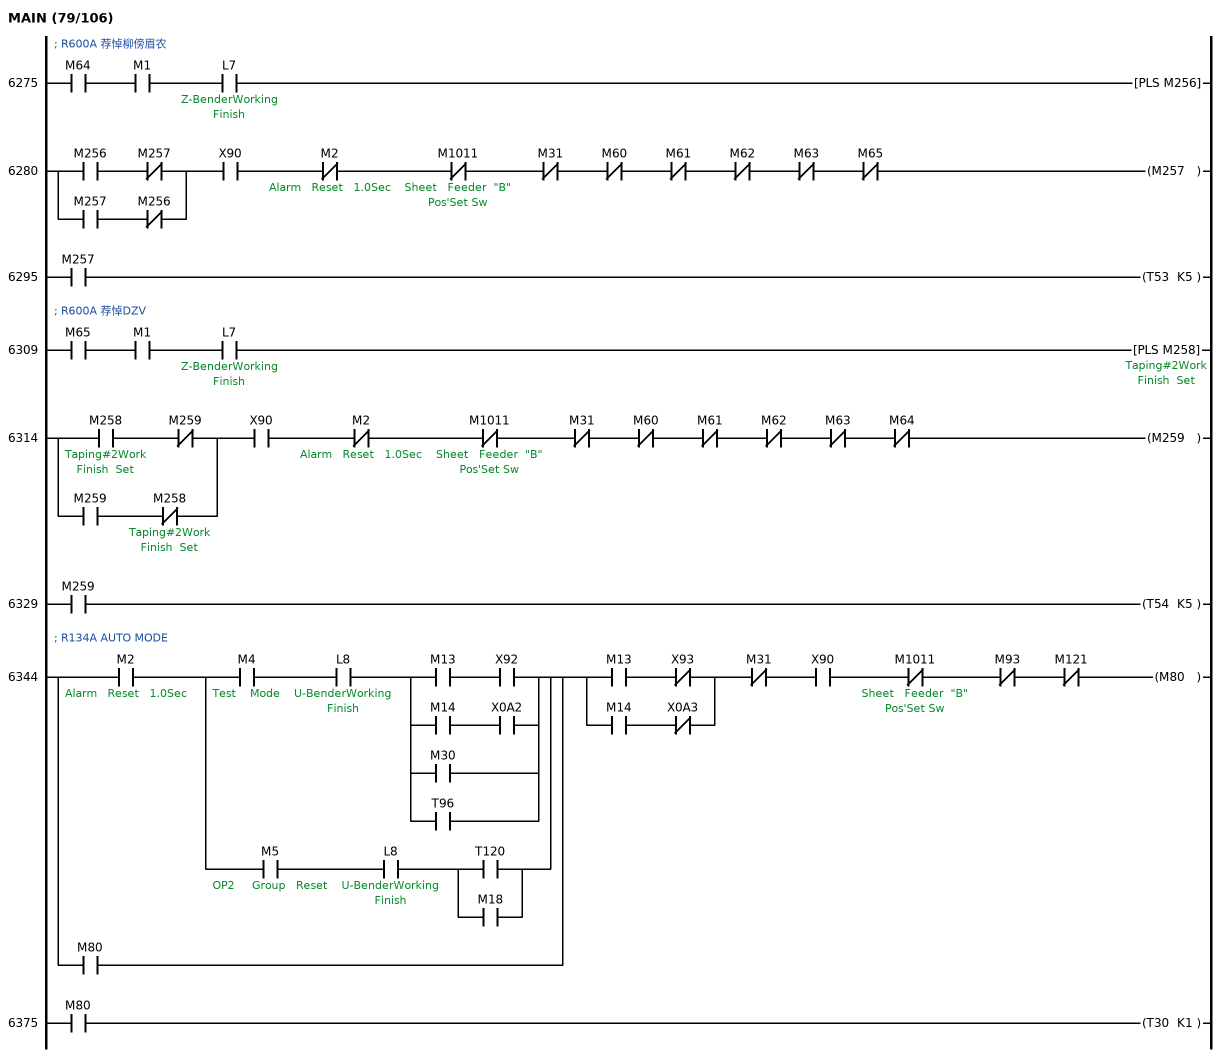
; R600A 수동진공체크
6275  LD      M64
      AND     M1
      AND     L7  ; Z-BenderWorking Finish
      PLS     M256
6280  LD      M256
      ANI     M257
      LD      M257
      ANI     M256
      ORB
      AND     X90
      ANI     M2  ; Alarm   Reset   1.0Sec
      ANI     M1011  ; Sheet   Feeder  "B" Pos'Set Sw
      ANI     M31
      ANI     M60
      ANI     M61
      ANI     M62
      ANI     M63
      ANI     M65
      OUT     M257
6295  LD      M257
      OUT     T53 K5
; R600A 수동DZV
6309  LD      M65
      AND     M1
      AND     L7  ; Z-BenderWorking Finish
      PLS     M258  ; Taping#2Work    Finish  Set
6314  LD      M258  ; Taping#2Work    Finish  Set
      ANI     M259
      LD      M259
      ANI     M258  ; Taping#2Work    Finish  Set
      ORB
      AND     X90
      ANI     M2  ; Alarm   Reset   1.0Sec
      ANI     M1011  ; Sheet   Feeder  "B" Pos'Set Sw
      ANI     M31
      ANI     M60
      ANI     M61
      ANI     M62
      ANI     M63
      ANI     M64
      OUT     M259
6329  LD      M259
      OUT     T54 K5
; R134A AUTO MODE
6344  LD      M2  ; Alarm   Reset   1.0Sec
      LD      M4  ; Test    Mode
      AND     L8  ; U-BenderWorking Finish
      LD      M13
      AND     X92
      LD      M14
      AND     X0A2
      ORB
      OR      M30
      OR      T96
      ANB
      LD      M5  ; OP2     Group   Reset
      AND     L8  ; U-BenderWorking Finish
      LD      T120
      OR      M18
      ANB
      ORB
      ANB
      OR      M80
      LD      M13
      ANI     X93
      LD      M14
      ANI     X0A3
      ORB
      ANB
      ANI     M31
      AND     X90
      ANI     M1011  ; Sheet   Feeder  "B" Pos'Set Sw
      ANI     M93
      ANI     M121
      OUT     M80
6375  LD      M80
      OUT     T30 K1
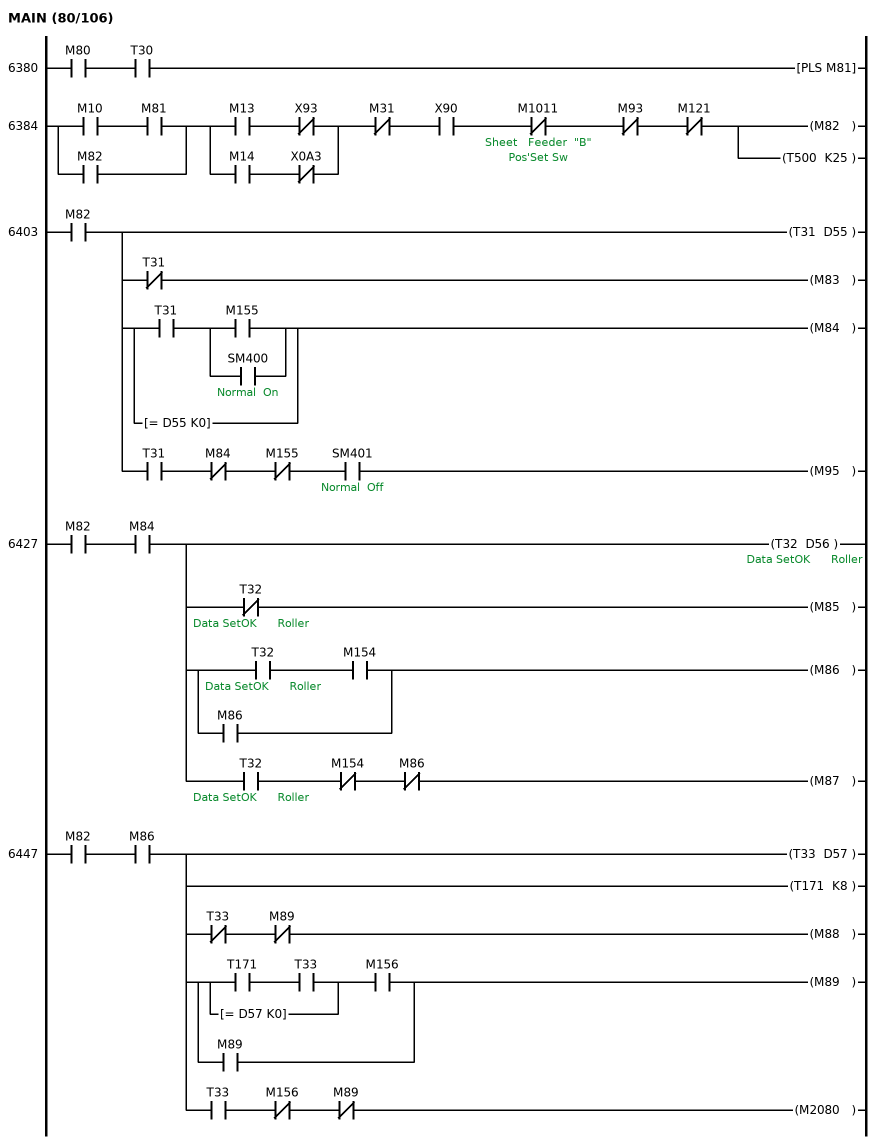
6380  LD      M80
      AND     T30
      PLS     M81
6384  LD      M10
      AND     M81
      OR      M82
      LD      M13
      ANI     X93
      LD      M14
      ANI     X0A3
      ORB
      ANB
      ANI     M31
      AND     X90
      ANI     M1011  ; Sheet   Feeder  "B" Pos'Set Sw
      ANI     M93
      ANI     M121
      OUT     M82
      OUT     T500 K25
6403  LD      M82
      OUT     T31 D55
      MPS
      ANI     T31
      OUT     M83
      MRD
      LD      T31
      LD      M155
      OR      SM400  ; Normal  On
      ANB
      OR=     D55 K0
      ANB
      OUT     M84
      MPP
      AND     T31
      ANI     M84
      ANI     M155
      AND     SM401  ; Normal  Off
      OUT     M95
6427  LD      M82
      AND     M84
      OUT     T32 D56  ; Data SetOK      Roller
      MPS
      ANI     T32  ; Data SetOK      Roller
      OUT     M85
      MRD
      LD      T32  ; Data SetOK      Roller
      AND     M154
      OR      M86
      ANB
      OUT     M86
      MPP
      AND     T32  ; Data SetOK      Roller
      ANI     M154
      ANI     M86
      OUT     M87
6447  LD      M82
      AND     M86
      OUT     T33 D57
      OUT     T171 K8
      MPS
      ANI     T33
      ANI     M89
      OUT     M88
      MRD
      LD      T171
      AND     T33
      OR=     D57 K0
      AND     M156
      OR      M89
      ANB
      OUT     M89
      MPP
      AND     T33
      ANI     M156
      ANI     M89
      OUT     M2080
